{attribute 'conditionalshow'}
FUNCTION_BLOCK FB_CV_BYTE_TO_WORD
VAR_INPUT
	{attribute 'hide'}
	byInputValue_1					: BYTE;								//Input value that is converted into the output value	
	{attribute 'hide'}						
	byInputValue_2					: BYTE;								//Input value that is converted into the output value
	{attribute 'hide'}
	eByteOrderForConvert			: eByteOrder;						//Byte Format
END_VAR
VAR_OUTPUT
	{attribute 'hide'}
	wOutputValue					: WORD;								//Converted output value
END_VAR
VAR
END_VAR

//Creator : Kai Ebensperger
//Company : Lynus AG
//Date : 28.04.2021
//Version : 1.0.0.0

//With this functionblock its possible to convert a certain Datatyp in a other Datatype
//The byte order can be selected between BigEndian and LittleEndian
//BYTE TO WORD
//Created for the Edge Device Lib over Modbus TCP
//Modbus TCP is WORD oriented

IF eByteOrderForConvert = eByteOrder.eBigEndian THEN
	wOutputValue := SHL(BYTE_TO_WORD(byInputValue_1),8) + BYTE_TO_WORD(byInputValue_2);
ELSE
	wOutputValue := SHL(BYTE_TO_WORD(byInputValue_2),8) + BYTE_TO_WORD(byInputValue_1);
END_IF

END_FUNCTION_BLOCK

(* stored: Version 1.1.0.1, ProductVersion 3.1.4024.9
   POU FB_CV_BYTE_TO_WORD: Id {366295f6-72cd-4be4-a77e-c8ce56e2952b}, SpecialFunc None *)
